// TIA Portal V20 export
// export: Created 2025-12-01T14:56:48.18536Z, ExportSetting None, DisplayName Totally Integrated Automation Portal, DisplayVersion V20 Update 3, DisplayName TIA Portal Openness, DisplayVersion V20 Update 3, DisplayName TIA Portal Version Control Interface, DisplayVersion V20 Update 3, DisplayName STEP 7 Professional, DisplayVersion V20 Update 3, DisplayName STEP 7 Safety, DisplayVersion V20 Update 2, DisplayName WinCC Basic/Comfort/Advanced, DisplayVersion V20 Update 3, DisplayName WinCC Professional, DisplayVersion V20 Update 3, DisplayName WinCC Unified, DisplayVersion V20 Update 3
FUNCTION_BLOCK "FB91_MLG_SICK_ALTURA_V02"   // FB91, LAD
{ S7_Optimized_Access := 'FALSE' }
// stored: AutoNumber false, SetENOAutomatically false
   VAR_INPUT
      NBB : Int;
      Barrera_Word02 : Int;
      Barrera_Word03 : Int;
      Resolucion : Int;
      Offset : Int;
      ActivarLectura : Bool;
   END_VAR
   VAR_OUTPUT
      AlturaBulto : Int;
   END_VAR
   VAR
      MemoriaAlturaBulto : Int;
      AlturaActual { ExternalVisible := 'False'} : Int;
      AlturaLeida_Puntos { ExternalVisible := 'False'} : Int;
   END_VAR
   VAR_TEMP
      NuevaAltura : Int;
      DatoValido : Bool;
   END_VAR
BEGIN

NETWORK
TITLE = Inicializar
// -----------------------------------------------------------------------
// --- Inicializar

      L     #NBB;  // Altura Leida (Puntos)
      T     #AlturaLeida_Puntos;


      A     #ActivarLectura;
      JC    LeerAltura;

      L     0;
      T     #MemoriaAlturaBulto;

      JU    FinFuncion;



NETWORK
TITLE = Leer la Altura
// -----------------------------------------------------------------------
// --- Mirar si hay Lectura Nueva
// --- Byte 01  Bit 0 y Bit 1 uno de los dos a uno
// ---          Bit 2 Dato Valido

LeerAltura:NOP   0;
      L     #AlturaLeida_Puntos;
      L     0;
      <>I;
      =     #DatoValido;

      AN    #DatoValido;
      JC    FinFuncion;




NETWORK
TITLE = Calcular Altura
// -----------------------------------------------------------------------
// --- Calcula la Altura Actual
// --- NuevaAltura = (LeidoAltura * Resolucion) + Offset

      L     #AlturaLeida_Puntos;
      L     #Resolucion;
      *I;
      L     #Offset;
      +I;
      T     #NuevaAltura;


// -----------------------------------------------------------------------
// --- Comprobar si es Mayor que la Nueva

      L     #NuevaAltura;  // Si la Altura Nueva
      L     #MemoriaAlturaBulto;  // Es Mayor o Igual
      >=I;
      JCN   FinFuncion;

      L     #AlturaActual;  // Gurado la Nueva Altura
      T     #MemoriaAlturaBulto;


NETWORK
TITLE = Final
// -----------------------------------------------------------------------
// --- Se Acabo. Dar la Altura Memorizada

FinFuncion:NOP   0;

      L     #MemoriaAlturaBulto;  // Altura Maxima Leida
      T     #AlturaBulto;

      L     #AlturaLeida_Puntos;  // Altura Actual
      L     #Resolucion;
      *I;
      L     #Offset;
      +I;
      T     #AlturaActual;

END_FUNCTION_BLOCK
